FUNCTION FF_BLOCK : REAL
VAR_INPUT
	input_value: REAL;
	k_ff: REAL;
END_VAR
VAR
END_VAR

FF_BLOCK := input_value * (1 + k_ff);

END_FUNCTION

(* stored: Version 1.1.0.1, ProductVersion 3.1.4024.15
   POU FF_BLOCK: Id {cf0c61b7-5dac-4ee3-9cb6-99bf0ae70e1d}, SpecialFunc None *)
